// TIA Portal V17 export
// export: Created 2026-04-13T11:12:44.6467311Z, ExportSetting WithDefaults, DisplayName Totally Integrated Automation Portal, DisplayVersion V17 Update 4, DisplayName TIA Portal Openness, DisplayVersion V17 Update 4, DisplayName TIA Portal Version Control Interface, DisplayVersion V17, DisplayName SINAMICS Startdrive Advanced, DisplayVersion V17, DisplayName SINAMICS Startdrive G130, G150, S120, S150, SINAMICS MV, S210, DisplayVersion V17, DisplayName SINAMICS Startdrive G110M, G120, G120C, G120D, G120P, G115D, DisplayVersion V17, DisplayName STEP 7 Professional, DisplayVersion V17 Update 4, DisplayName STEP 7 Safety, DisplayVersion V17, DisplayName WinCC Professional, DisplayVersion V17 Update 4
DATA_BLOCK "D2-室外CIP通讯_DB"   // DB35
VERSION : 0.1
// stored: AutoNumber true, DBAccessibleFromOPCUA true, DBAccessibleFromWebserver true, InstanceOfName D2-室外CIP通讯, InstanceOfType FB
"D2-室外CIP通讯"
   // VAR
   //    T_10HZ { S7_SetPoint := 'True'} : TON_TIME;
   //    FT1 { S7_SetPoint := 'True'} : F_TRIG;
   //    RT00 { S7_SetPoint := 'True'} : R_TRIG;
   //    RT10 { S7_SetPoint := 'True'} : R_TRIG;
   //    RT11 { S7_SetPoint := 'True'} : R_TRIG;
   //    RT12 { S7_SetPoint := 'True'} : R_TRIG;
   //    RT20 { S7_SetPoint := 'True'} : R_TRIG;
   //    RT21 { S7_SetPoint := 'True'} : R_TRIG;
   //    RT22 { S7_SetPoint := 'True'} : R_TRIG;
   //    RT30 { S7_SetPoint := 'True'} : R_TRIG;
   //    RT31 { S7_SetPoint := 'True'} : R_TRIG;
   //    RT32 { S7_SetPoint := 'True'} : R_TRIG;
   //    RT40 { S7_SetPoint := 'True'} : R_TRIG;
   //    RT41 { S7_SetPoint := 'True'} : R_TRIG;
   //    RT42 { S7_SetPoint := 'True'} : R_TRIG;
   //    RT50 { S7_SetPoint := 'True'} : R_TRIG;
   //    RT51 { S7_SetPoint := 'True'} : R_TRIG;
   //    RT60 { S7_SetPoint := 'True'} : R_TRIG;
   //    RT61 { S7_SetPoint := 'True'} : R_TRIG;
   //    RT62 { S7_SetPoint := 'True'} : R_TRIG;
   //    RT3 { S7_SetPoint := 'True'} : R_TRIG;
   //    RS热水洗辅助 { S7_SetPoint := 'True'} : Bool;
   //    JS碱水洗辅助 : Bool;
   //    CS纯水洗辅助 : Bool;
   //    EC二纯水洗辅助 : Bool;
   //    RJ溶剂洗辅助 : Bool;
   //    PUT_Instance { S7_SetPoint := 'True'} : PUT;
   //    GET_Instance { S7_SetPoint := 'True'} : GET;
   // END_VAR
BEGIN
END_DATA_BLOCK
